SYSTEM NEWQuestion2V_CNV_V2 (* System Configuration *)
  (* Standard: 61499-1 *)
  (* Version 0.4, 2009-03-05, JHC, Holobloc Inc., Deleted Application. *)
  (* Version 0.3, 2003-12-05, JHC, Rockwell Automation, Renamed from NEWSYSTEM. *)
  (* Version 0.2, 2002-11-05, JHC, Rockwell Automation, Fixed missing (empty) FBD in Application. *)
  (* Version 0.1, 2002-01-17, JHC, Rockwell Automation, Minor cleanup *)
  (* Version 0.0, 2000-05-27, JHC, Rockwell Automation *)
  DEVICE HMI : FRAME_DEVICE(GRID := [6,1], BOUNDS := [810,10,300,300])
    RESOURCE reset : PANEL_RESOURCE
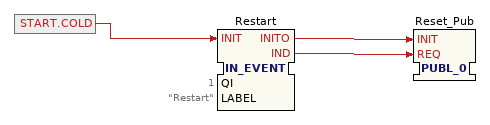
      FBS
        Restart : IN_EVENT(QI := 1, LABEL := "Restart");
        Reset_Pub : PUBL_0;
      END_FBS
      EVENT_CONNECTIONS
        START.COLD TO Restart.INIT;
        Restart.INITO TO Reset_Pub.INIT;
        Restart.IND TO Reset_Pub.REQ;
      END_CONNECTIONS
    END_RESOURCE
    RESOURCE motor_1 : PANEL_RESOURCE
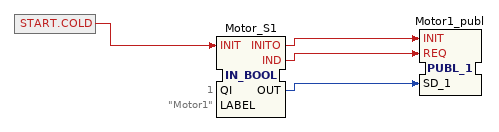
      FBS
        Motor_S1 : IN_BOOL(QI := 1, LABEL := "Motor1");
        Motor1_publ : PUBL_1;
      END_FBS
      EVENT_CONNECTIONS
        START.COLD TO Motor_S1.INIT;
        Motor_S1.INITO TO Motor1_publ.INIT;
        Motor_S1.IND TO Motor1_publ.REQ;
      END_CONNECTIONS
      DATA_CONNECTIONS
        Motor_S1.OUT TO Motor1_publ.SD_1;
      END_CONNECTIONS
    END_RESOURCE
    RESOURCE motor2 : PANEL_RESOURCE
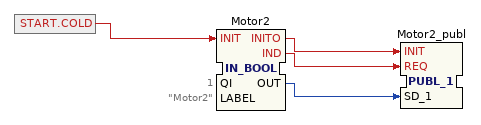
      FBS
        Motor2 : IN_BOOL(QI := 1, LABEL := "Motor2");
        Motor2_publ : PUBL_1;
      END_FBS
      EVENT_CONNECTIONS
        START.COLD TO Motor2.INIT;
        Motor2.INITO TO Motor2_publ.INIT;
        Motor2.IND TO Motor2_publ.REQ;
      END_CONNECTIONS
      DATA_CONNECTIONS
        Motor2.OUT TO Motor2_publ.SD_1;
      END_CONNECTIONS
    END_RESOURCE
    RESOURCE motor3_red : PANEL_RESOURCE
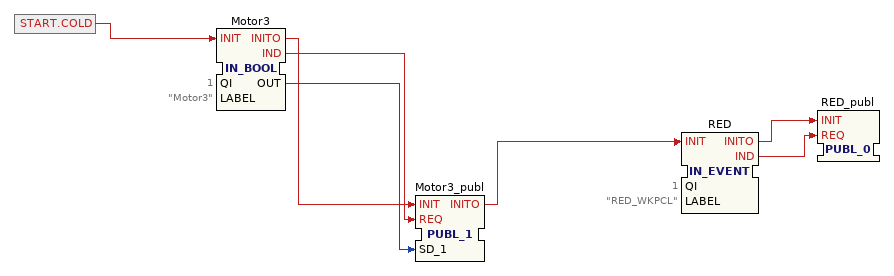
      FBS
        Motor3_publ : PUBL_1;
        Motor3 : IN_BOOL(QI := 1, LABEL := "Motor3");
        RED : IN_EVENT(QI := 1, LABEL := "RED_WKPCL");
        RED_publ : PUBL_0;
      END_FBS
      EVENT_CONNECTIONS
        START.COLD TO Motor3.INIT;
        Motor3.INITO TO Motor3_publ.INIT;
        Motor3.IND TO Motor3_publ.REQ;
        Motor3_publ.INITO TO RED.INIT;
        RED.INITO TO RED_publ.INIT;
        RED.IND TO RED_publ.REQ;
      END_CONNECTIONS
      DATA_CONNECTIONS
        Motor3.OUT TO Motor3_publ.SD_1;
      END_CONNECTIONS
    END_RESOURCE
    RESOURCE motor4_yellow : PANEL_RESOURCE
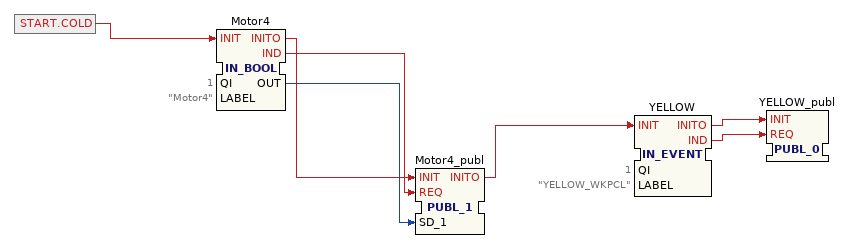
      FBS
        Motor4_publ : PUBL_1;
        Motor4 : IN_BOOL(QI := 1, LABEL := "Motor4");
        YELLOW : IN_EVENT(QI := 1, LABEL := "YELLOW_WKPCL");
        YELLOW_publ : PUBL_0;
      END_FBS
      EVENT_CONNECTIONS
        START.COLD TO Motor4.INIT;
        Motor4.INITO TO Motor4_publ.INIT;
        Motor4.IND TO Motor4_publ.REQ;
        Motor4_publ.INITO TO YELLOW.INIT;
        YELLOW.INITO TO YELLOW_publ.INIT;
        YELLOW.IND TO YELLOW_publ.REQ;
      END_CONNECTIONS
      DATA_CONNECTIONS
        Motor4.OUT TO Motor4_publ.SD_1;
      END_CONNECTIONS
    END_RESOURCE
    RESOURCE motor5_blue : PANEL_RESOURCE
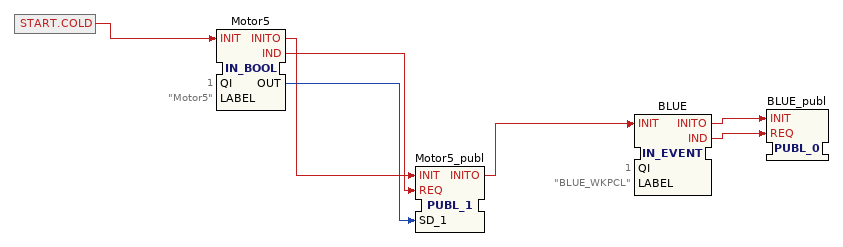
      FBS
        Motor5_publ : PUBL_1;
        Motor5 : IN_BOOL(QI := 1, LABEL := "Motor5");
        BLUE : IN_EVENT(QI := 1, LABEL := "BLUE_WKPCL");
        BLUE_publ : PUBL_0;
      END_FBS
      EVENT_CONNECTIONS
        START.COLD TO Motor5.INIT;
        Motor5.INITO TO Motor5_publ.INIT;
        Motor5.IND TO Motor5_publ.REQ;
        Motor5_publ.INITO TO BLUE.INIT;
        BLUE.INITO TO BLUE_publ.INIT;
        BLUE.IND TO BLUE_publ.REQ;
      END_CONNECTIONS
      DATA_CONNECTIONS
        Motor5.OUT TO Motor5_publ.SD_1;
      END_CONNECTIONS
    END_RESOURCE
  END_DEVICE
  DEVICE VIEW : FRAME_DEVICE(BOUNDS := [10,10,500,700], GRID := [1,1])
    RESOURCE CNV : PANEL_RESOURCE
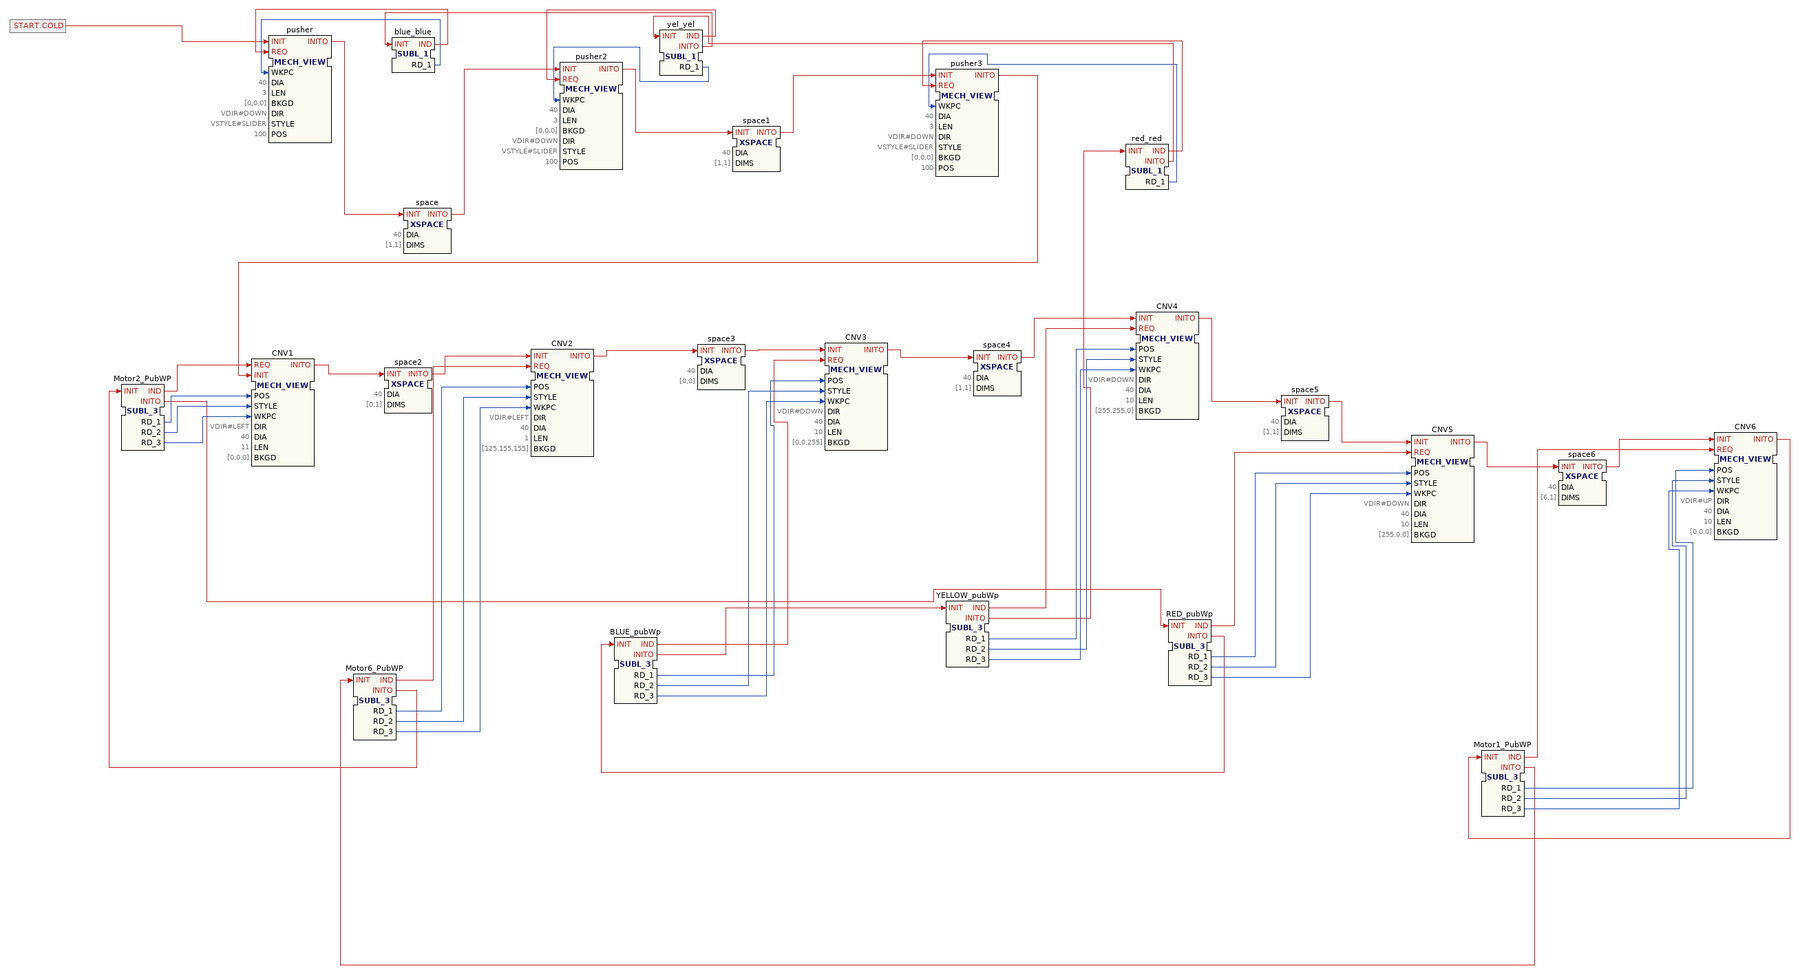
      FBS
        CNV1 : MECH_VIEW(DIR := VDIR#LEFT, DIA := 40, LEN := 11, BKGD := [0,0,0]);
        CNV2 : MECH_VIEW(DIR := VDIR#LEFT, DIA := 40, LEN := 1, BKGD := [125,155,155]);
        CNV3 : MECH_VIEW(DIR := VDIR#DOWN, DIA := 40, LEN := 10, BKGD := [0,0,255]);
        CNV4 : MECH_VIEW(DIR := VDIR#DOWN, DIA := 40, LEN := 10, BKGD := [255,255,0]);
        CNV5 : MECH_VIEW(DIR := VDIR#DOWN, DIA := 40, LEN := 10, BKGD := [255,0,0]);
        CNV6 : MECH_VIEW(DIR := VDIR#UP, DIA := 40, LEN := 10, BKGD := [0,0,0]);
        space2 : XSPACE(DIA := 40, DIMS := [0,1]);
        space3 : XSPACE(DIA := 40, DIMS := [0,0]);
        space4 : XSPACE(DIA := 40, DIMS := [1,1]);
        space5 : XSPACE(DIA := 40, DIMS := [1,1]);
        space6 : XSPACE(DIA := 40, DIMS := [6,1]);
        space : XSPACE(DIA := 40, DIMS := [1,1]);
        space1 : XSPACE(DIA := 40, DIMS := [1,1]);
        Motor1_PubWP : SUBL_3;
        Motor6_PubWP : SUBL_3;
        Motor2_PubWP : SUBL_3;
        BLUE_pubWp : SUBL_3;
        YELLOW_pubWp : SUBL_3;
        RED_pubWp : SUBL_3;
        pusher : MECH_VIEW(DIA := 40, LEN := 3, BKGD := [0,0,0], DIR := VDIR#DOWN, STYLE := VSTYLE#SLIDER, POS := 100);
        pusher2 : MECH_VIEW(DIA := 40, LEN := 3, BKGD := [0,0,0], DIR := VDIR#DOWN, STYLE := VSTYLE#SLIDER, POS := 100);
        pusher3 : MECH_VIEW(DIA := 40, LEN := 3, DIR := VDIR#DOWN, STYLE := VSTYLE#SLIDER, BKGD := [0,0,0], POS := 100);
        red_red : SUBL_1;
        yel_yel : SUBL_1;
        blue_blue : SUBL_1;
      END_FBS
      EVENT_CONNECTIONS
        CNV1.INITO TO space2.INIT;
        space2.INITO TO CNV2.INIT;
        CNV2.INITO TO space3.INIT;
        space3.INITO TO CNV3.INIT;
        CNV3.INITO TO space4.INIT;
        space4.INITO TO CNV4.INIT;
        CNV4.INITO TO space5.INIT;
        space5.INITO TO CNV5.INIT;
        CNV5.INITO TO space6.INIT;
        space6.INITO TO CNV6.INIT;
        CNV6.INITO TO Motor1_PubWP.INIT;
        Motor1_PubWP.IND TO CNV6.REQ;
        Motor1_PubWP.INITO TO Motor6_PubWP.INIT;
        Motor6_PubWP.IND TO CNV2.REQ;
        Motor6_PubWP.INITO TO Motor2_PubWP.INIT;
        Motor2_PubWP.IND TO CNV1.REQ;
        BLUE_pubWp.IND TO CNV3.REQ;
        BLUE_pubWp.INITO TO YELLOW_pubWp.INIT;
        YELLOW_pubWp.IND TO CNV4.REQ;
        RED_pubWp.IND TO CNV5.REQ;
        Motor2_PubWP.INITO TO RED_pubWp.INIT;
        RED_pubWp.INITO TO BLUE_pubWp.INIT;
        START.COLD TO pusher.INIT;
        pusher.INITO TO space.INIT;
        space.INITO TO pusher2.INIT;
        pusher2.INITO TO space1.INIT;
        space1.INITO TO pusher3.INIT;
        pusher3.INITO TO CNV1.INIT;
        red_red.IND TO pusher3.REQ;
        YELLOW_pubWp.INITO TO red_red.INIT;
        red_red.INITO TO yel_yel.INIT;
        yel_yel.IND TO pusher2.REQ;
        yel_yel.INITO TO blue_blue.INIT;
        blue_blue.IND TO pusher.REQ;
      END_CONNECTIONS
      DATA_CONNECTIONS
        Motor1_PubWP.RD_1 TO CNV6.POS;
        Motor1_PubWP.RD_2 TO CNV6.STYLE;
        Motor1_PubWP.RD_3 TO CNV6.WKPC;
        Motor6_PubWP.RD_1 TO CNV2.POS;
        Motor6_PubWP.RD_2 TO CNV2.STYLE;
        Motor6_PubWP.RD_3 TO CNV2.WKPC;
        Motor2_PubWP.RD_1 TO CNV1.POS;
        Motor2_PubWP.RD_2 TO CNV1.STYLE;
        Motor2_PubWP.RD_3 TO CNV1.WKPC;
        BLUE_pubWp.RD_1 TO CNV3.POS;
        BLUE_pubWp.RD_2 TO CNV3.STYLE;
        BLUE_pubWp.RD_3 TO CNV3.WKPC;
        YELLOW_pubWp.RD_1 TO CNV4.POS;
        YELLOW_pubWp.RD_2 TO CNV4.STYLE;
        YELLOW_pubWp.RD_3 TO CNV4.WKPC;
        RED_pubWp.RD_1 TO CNV5.POS;
        RED_pubWp.RD_2 TO CNV5.STYLE;
        RED_pubWp.RD_3 TO CNV5.WKPC;
        red_red.RD_1 TO pusher3.WKPC;
        yel_yel.RD_1 TO pusher2.WKPC;
        blue_blue.RD_1 TO pusher.WKPC;
      END_CONNECTIONS
    END_RESOURCE
  END_DEVICE
  DEVICE MODEL : FRAME_DEVICE(BOUNDS := [0,0,0,0], GRID := [1,1])
    RESOURCE CLK : PANEL_RESOURCE
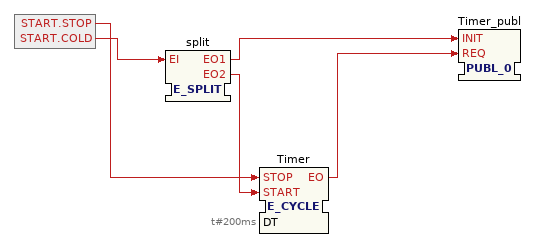
      FBS
        Timer : E_CYCLE(DT := t#200ms);
        Timer_publ : PUBL_0;
        split : E_SPLIT;
      END_FBS
      EVENT_CONNECTIONS
        START.STOP TO Timer.STOP;
        START.COLD TO split.EI;
        split.EO1 TO Timer_publ.INIT;
        split.EO2 TO Timer.START;
        Timer.EO TO Timer_publ.REQ;
      END_CONNECTIONS
    END_RESOURCE
    RESOURCE Motor1 : PANEL_RESOURCE
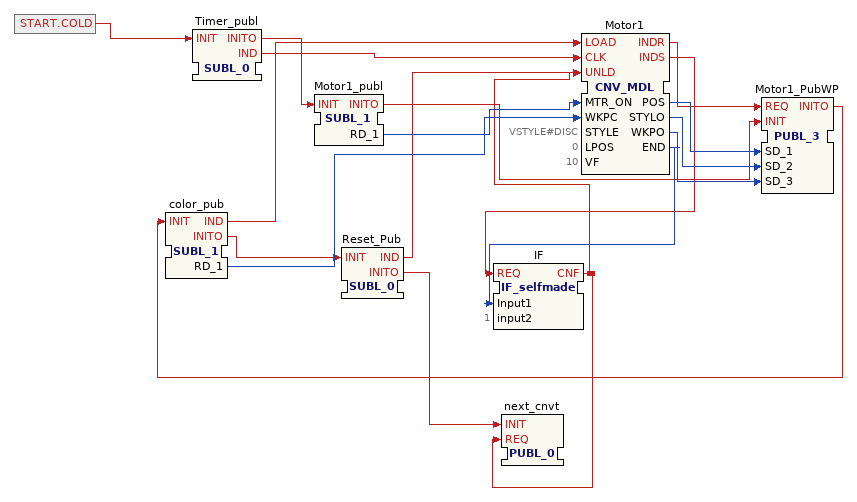
      FBS
        Timer_publ : SUBL_0;
        Motor1_publ : SUBL_1;
        Motor1 : CNV_MDL(STYLE := VSTYLE#DISC, LPOS := 0, VF := 10);
        Motor1_PubWP : PUBL_3;
        color_pub : SUBL_1;
        Reset_Pub : SUBL_0;
        IF : IF_selfmade(input2 := 1);
        next_cnvt : PUBL_0;
      END_FBS
      EVENT_CONNECTIONS
        START.COLD TO Timer_publ.INIT;
        Timer_publ.INITO TO Motor1_publ.INIT;
        Motor1.INDR TO Motor1_PubWP.REQ;
        Motor1_publ.INITO TO Motor1_PubWP.INIT;
        Motor1_PubWP.INITO TO color_pub.INIT;
        color_pub.IND TO Motor1.LOAD;
        Timer_publ.IND TO Motor1.CLK;
        color_pub.INITO TO Reset_Pub.INIT;
        Reset_Pub.IND TO Motor1.UNLD;
        Motor1.INDS TO IF.REQ;
        IF.CNF TO Motor1.UNLD;
        Reset_Pub.INITO TO next_cnvt.INIT;
        IF.CNF TO next_cnvt.REQ;
      END_CONNECTIONS
      DATA_CONNECTIONS
        Motor1_publ.RD_1 TO Motor1.MTR_ON;
        Motor1.POS TO Motor1_PubWP.SD_1;
        Motor1.STYLO TO Motor1_PubWP.SD_2;
        Motor1.WKPO TO Motor1_PubWP.SD_3;
        color_pub.RD_1 TO Motor1.WKPC;
        Motor1.END TO IF.Input1;
      END_CONNECTIONS
    END_RESOURCE
    RESOURCE motor2 : PANEL_RESOURCE
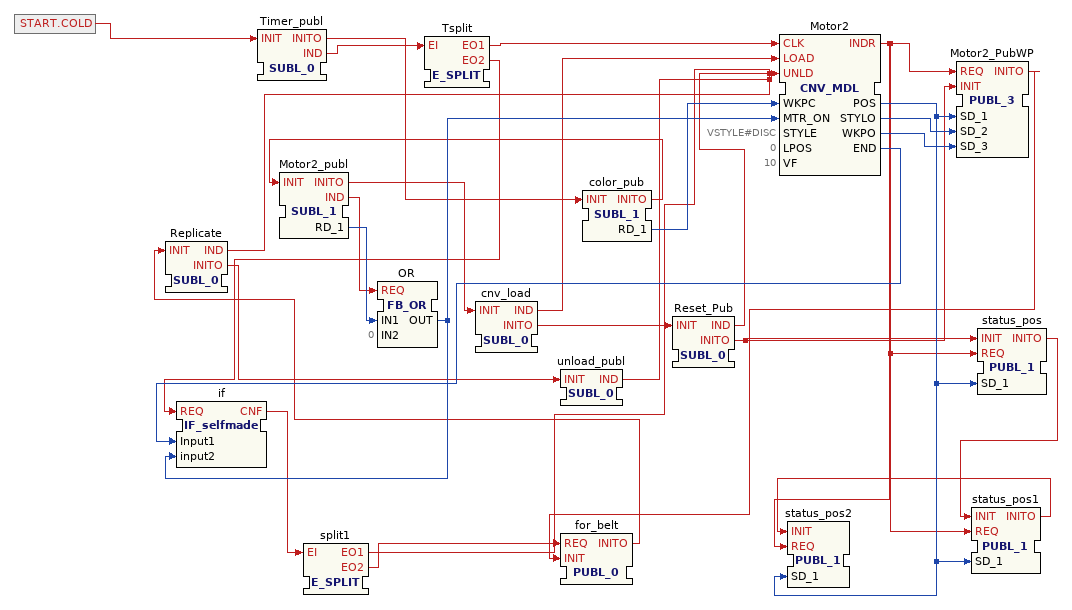
      FBS
        Motor2 : CNV_MDL(STYLE := VSTYLE#DISC, LPOS := 0, VF := 10);
        Timer_publ : SUBL_0;
        Tsplit : E_SPLIT;
        color_pub : SUBL_1;
        Motor2_publ : SUBL_1;
        cnv_load : SUBL_0;
        Motor2_PubWP : PUBL_3;
        Reset_Pub : SUBL_0;
        split1 : E_SPLIT;
        if : IF_selfmade;
        OR : FB_OR(IN2 := 0);
        for_belt : PUBL_0;
        Replicate : SUBL_0;
        unload_publ : SUBL_0;
        status_pos : PUBL_1;
        status_pos1 : PUBL_1;
        status_pos2 : PUBL_1;
      END_FBS
      EVENT_CONNECTIONS
        START.COLD TO Timer_publ.INIT;
        Tsplit.EO1 TO Motor2.CLK;
        color_pub.INITO TO Motor2_publ.INIT;
        Motor2_publ.INITO TO cnv_load.INIT;
        cnv_load.IND TO Motor2.LOAD;
        Timer_publ.INITO TO color_pub.INIT;
        Reset_Pub.IND TO Motor2.UNLD;
        Motor2.INDR TO Motor2_PubWP.REQ;
        Reset_Pub.INITO TO Motor2_PubWP.INIT;
        split1.EO1 TO Motor2.UNLD;
        if.CNF TO split1.EI;
        Motor2_publ.IND TO OR.REQ;
        cnv_load.INITO TO Reset_Pub.INIT;
        Tsplit.EO2 TO if.REQ;
        split1.EO2 TO for_belt.REQ;
        Motor2_PubWP.INITO TO for_belt.INIT;
        Timer_publ.IND TO Tsplit.EI;
        Replicate.IND TO Motor2.UNLD;
        for_belt.INITO TO Replicate.INIT;
        unload_publ.IND TO Motor2.UNLD;
        Replicate.INITO TO unload_publ.INIT;
        Reset_Pub.INITO TO status_pos.INIT;
        Motor2.INDR TO status_pos.REQ;
        status_pos.INITO TO status_pos1.INIT;
        Motor2.INDR TO status_pos1.REQ;
        status_pos1.INITO TO status_pos2.INIT;
        Motor2.INDR TO status_pos2.REQ;
      END_CONNECTIONS
      DATA_CONNECTIONS
        color_pub.RD_1 TO Motor2.WKPC;
        Motor2.POS TO Motor2_PubWP.SD_1;
        Motor2.STYLO TO Motor2_PubWP.SD_2;
        Motor2.WKPO TO Motor2_PubWP.SD_3;
        Motor2_publ.RD_1 TO OR.IN1;
        OR.OUT TO Motor2.MTR_ON;
        OR.OUT TO if.input2;
        Motor2.END TO if.Input1;
        Motor2.POS TO status_pos.SD_1;
        Motor2.POS TO status_pos1.SD_1;
        Motor2.POS TO status_pos2.SD_1;
      END_CONNECTIONS
    END_RESOURCE
    RESOURCE motor3_red : PANEL_RESOURCE
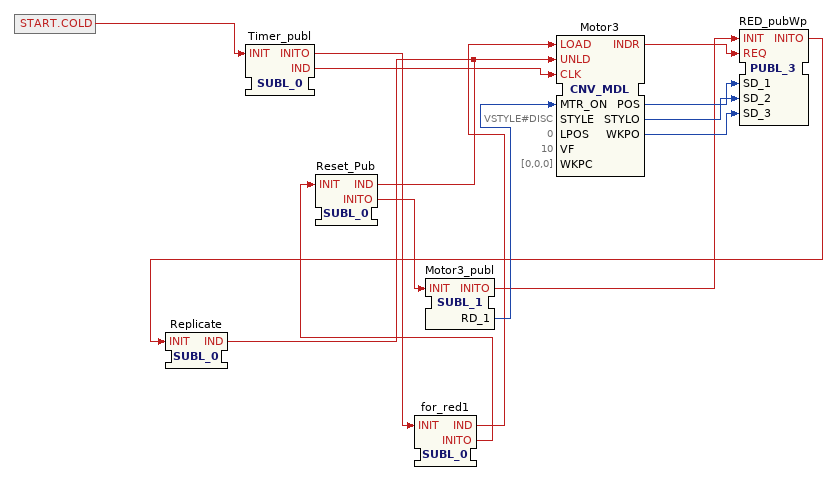
      FBS
        Timer_publ : SUBL_0;
        Motor3 : CNV_MDL(STYLE := VSTYLE#DISC, LPOS := 0, VF := 10, WKPC := [0,0,0]);
        for_red1 : SUBL_0;
        Reset_Pub : SUBL_0;
        Motor3_publ : SUBL_1;
        RED_pubWp : PUBL_3;
        Replicate : SUBL_0;
      END_FBS
      EVENT_CONNECTIONS
        START.COLD TO Timer_publ.INIT;
        Timer_publ.INITO TO for_red1.INIT;
        for_red1.IND TO Motor3.LOAD;
        for_red1.INITO TO Reset_Pub.INIT;
        Reset_Pub.IND TO Motor3.UNLD;
        Reset_Pub.INITO TO Motor3_publ.INIT;
        Motor3_publ.INITO TO RED_pubWp.INIT;
        Motor3.INDR TO RED_pubWp.REQ;
        Timer_publ.IND TO Motor3.CLK;
        RED_pubWp.INITO TO Replicate.INIT;
        Replicate.IND TO Motor3.UNLD;
      END_CONNECTIONS
      DATA_CONNECTIONS
        Motor3_publ.RD_1 TO Motor3.MTR_ON;
        Motor3.POS TO RED_pubWp.SD_1;
        Motor3.STYLO TO RED_pubWp.SD_2;
        Motor3.WKPO TO RED_pubWp.SD_3;
      END_CONNECTIONS
    END_RESOURCE
    RESOURCE motor4_yellow : PANEL_RESOURCE
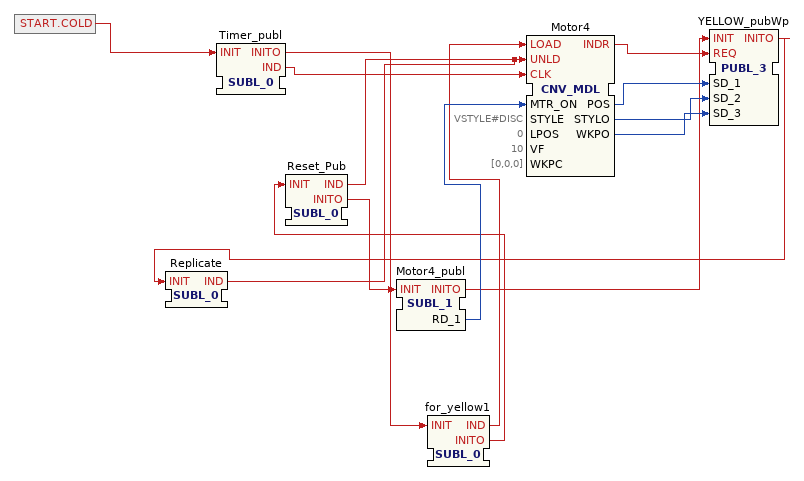
      FBS
        Timer_publ : SUBL_0;
        Motor4 : CNV_MDL(STYLE := VSTYLE#DISC, LPOS := 0, VF := 10, WKPC := [0,0,0]);
        for_yellow1 : SUBL_0;
        Reset_Pub : SUBL_0;
        Motor4_publ : SUBL_1;
        YELLOW_pubWp : PUBL_3;
        Replicate : SUBL_0;
      END_FBS
      EVENT_CONNECTIONS
        START.COLD TO Timer_publ.INIT;
        Timer_publ.INITO TO for_yellow1.INIT;
        for_yellow1.IND TO Motor4.LOAD;
        for_yellow1.INITO TO Reset_Pub.INIT;
        Reset_Pub.IND TO Motor4.UNLD;
        Reset_Pub.INITO TO Motor4_publ.INIT;
        Motor4_publ.INITO TO YELLOW_pubWp.INIT;
        Motor4.INDR TO YELLOW_pubWp.REQ;
        Timer_publ.IND TO Motor4.CLK;
        YELLOW_pubWp.INITO TO Replicate.INIT;
        Replicate.IND TO Motor4.UNLD;
      END_CONNECTIONS
      DATA_CONNECTIONS
        Motor4_publ.RD_1 TO Motor4.MTR_ON;
        Motor4.POS TO YELLOW_pubWp.SD_1;
        Motor4.STYLO TO YELLOW_pubWp.SD_2;
        Motor4.WKPO TO YELLOW_pubWp.SD_3;
      END_CONNECTIONS
    END_RESOURCE
    RESOURCE motor5_blue : PANEL_RESOURCE
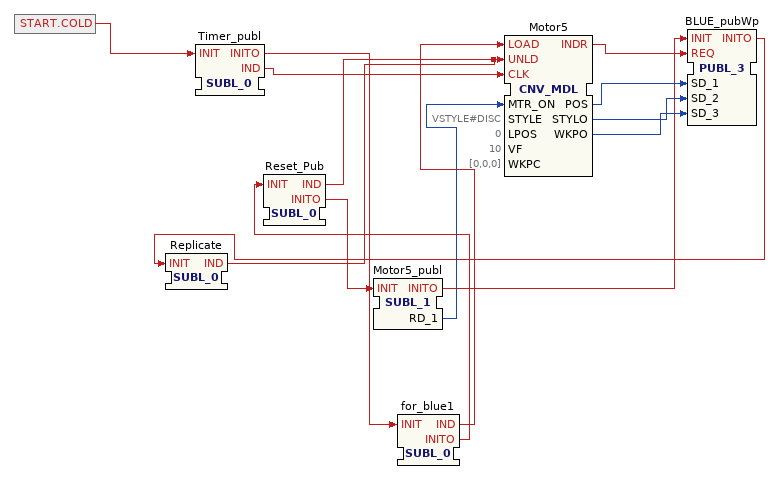
      FBS
        Timer_publ : SUBL_0;
        Motor5 : CNV_MDL(STYLE := VSTYLE#DISC, LPOS := 0, VF := 10, WKPC := [0,0,0]);
        for_blue1 : SUBL_0;
        Reset_Pub : SUBL_0;
        Motor5_publ : SUBL_1;
        BLUE_pubWp : PUBL_3;
        Replicate : SUBL_0;
      END_FBS
      EVENT_CONNECTIONS
        START.COLD TO Timer_publ.INIT;
        Timer_publ.INITO TO for_blue1.INIT;
        for_blue1.IND TO Motor5.LOAD;
        for_blue1.INITO TO Reset_Pub.INIT;
        Reset_Pub.IND TO Motor5.UNLD;
        Reset_Pub.INITO TO Motor5_publ.INIT;
        Motor5_publ.INITO TO BLUE_pubWp.INIT;
        Motor5.INDR TO BLUE_pubWp.REQ;
        Timer_publ.IND TO Motor5.CLK;
        BLUE_pubWp.INITO TO Replicate.INIT;
        Replicate.IND TO Motor5.UNLD;
      END_CONNECTIONS
      DATA_CONNECTIONS
        Motor5_publ.RD_1 TO Motor5.MTR_ON;
        Motor5.POS TO BLUE_pubWp.SD_1;
        Motor5.STYLO TO BLUE_pubWp.SD_2;
        Motor5.WKPO TO BLUE_pubWp.SD_3;
      END_CONNECTIONS
    END_RESOURCE
    RESOURCE motor6_turntable : PANEL_RESOURCE
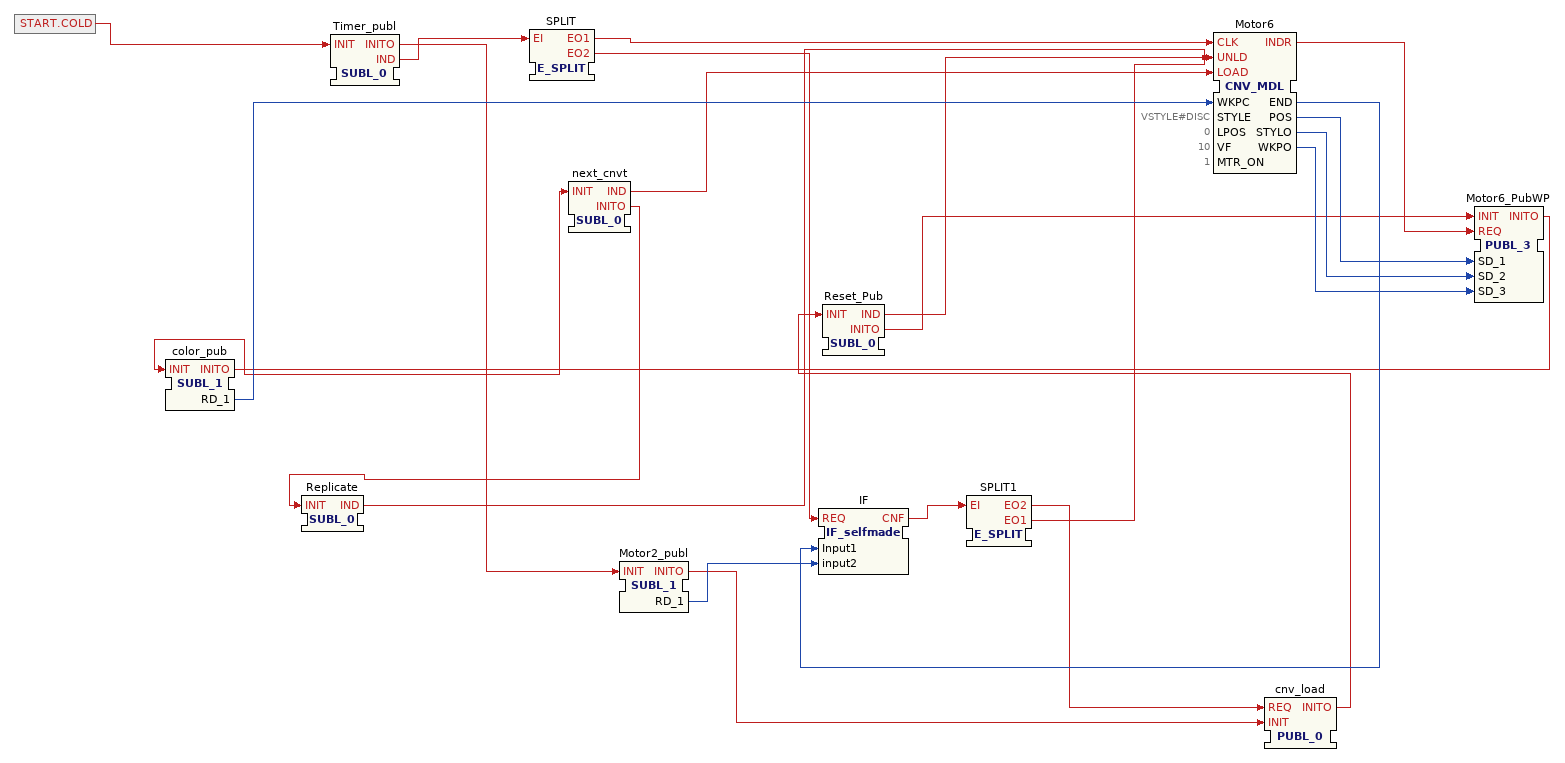
      FBS
        Motor6 : CNV_MDL(STYLE := VSTYLE#DISC, LPOS := 0, VF := 10, MTR_ON := 1);
        Timer_publ : SUBL_0;
        SPLIT : E_SPLIT;
        Motor2_publ : SUBL_1;
        IF : IF_selfmade;
        SPLIT1 : E_SPLIT;
        cnv_load : PUBL_0;
        Reset_Pub : SUBL_0;
        Motor6_PubWP : PUBL_3;
        color_pub : SUBL_1;
        next_cnvt : SUBL_0;
        Replicate : SUBL_0;
      END_FBS
      EVENT_CONNECTIONS
        START.COLD TO Timer_publ.INIT;
        SPLIT.EO1 TO Motor6.CLK;
        Timer_publ.INITO TO Motor2_publ.INIT;
        SPLIT.EO2 TO IF.REQ;
        IF.CNF TO SPLIT1.EI;
        SPLIT1.EO2 TO cnv_load.REQ;
        Motor2_publ.INITO TO cnv_load.INIT;
        cnv_load.INITO TO Reset_Pub.INIT;
        Reset_Pub.IND TO Motor6.UNLD;
        Reset_Pub.INITO TO Motor6_PubWP.INIT;
        Motor6.INDR TO Motor6_PubWP.REQ;
        Motor6_PubWP.INITO TO color_pub.INIT;
        color_pub.INITO TO next_cnvt.INIT;
        next_cnvt.IND TO Motor6.LOAD;
        Timer_publ.IND TO SPLIT.EI;
        SPLIT1.EO1 TO Motor6.UNLD;
        next_cnvt.INITO TO Replicate.INIT;
        Replicate.IND TO Motor6.UNLD;
      END_CONNECTIONS
      DATA_CONNECTIONS
        Motor6.END TO IF.Input1;
        Motor2_publ.RD_1 TO IF.input2;
        Motor6.POS TO Motor6_PubWP.SD_1;
        Motor6.STYLO TO Motor6_PubWP.SD_2;
        Motor6.WKPO TO Motor6_PubWP.SD_3;
        color_pub.RD_1 TO Motor6.WKPC;
      END_CONNECTIONS
    END_RESOURCE
  END_DEVICE
  DEVICE CONTROL : FRAME_DEVICE(BOUNDS := [0,0,0,0], GRID := [1,1])
    RESOURCE Color_control : PANEL_RESOURCE
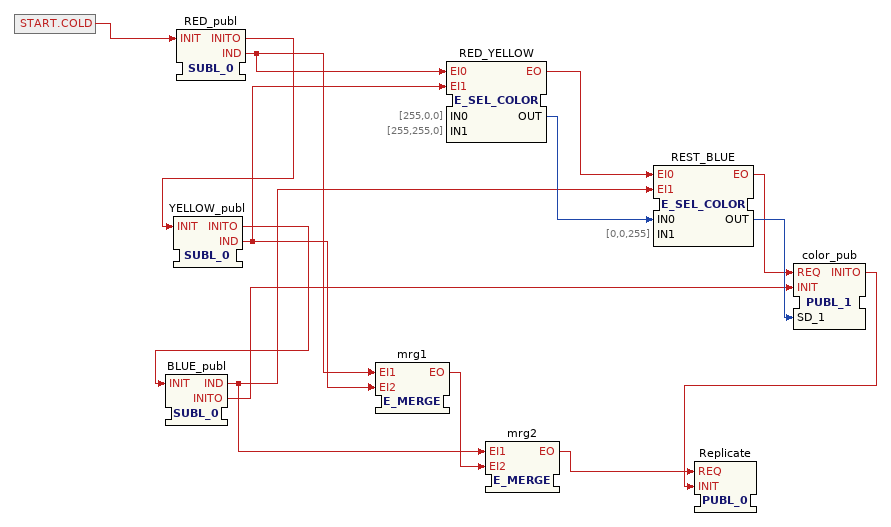
      FBS
        RED_publ : SUBL_0;
        YELLOW_publ : SUBL_0;
        BLUE_publ : SUBL_0;
        RED_YELLOW : E_SEL_COLOR(IN0 := [255,0,0], IN1 := [255,255,0]);
        REST_BLUE : E_SEL_COLOR(IN1 := [0,0,255]);
        color_pub : PUBL_1;
        mrg1 : E_MERGE;
        mrg2 : E_MERGE;
        Replicate : PUBL_0;
      END_FBS
      EVENT_CONNECTIONS
        START.COLD TO RED_publ.INIT;
        RED_publ.INITO TO YELLOW_publ.INIT;
        YELLOW_publ.INITO TO BLUE_publ.INIT;
        RED_publ.IND TO RED_YELLOW.EI0;
        YELLOW_publ.IND TO RED_YELLOW.EI1;
        RED_YELLOW.EO TO REST_BLUE.EI0;
        BLUE_publ.IND TO REST_BLUE.EI1;
        REST_BLUE.EO TO color_pub.REQ;
        BLUE_publ.INITO TO color_pub.INIT;
        RED_publ.IND TO mrg1.EI1;
        YELLOW_publ.IND TO mrg1.EI2;
        BLUE_publ.IND TO mrg2.EI1;
        mrg1.EO TO mrg2.EI2;
        mrg2.EO TO Replicate.REQ;
        color_pub.INITO TO Replicate.INIT;
      END_CONNECTIONS
      DATA_CONNECTIONS
        RED_YELLOW.OUT TO REST_BLUE.IN0;
        REST_BLUE.OUT TO color_pub.SD_1;
      END_CONNECTIONS
    END_RESOURCE
    RESOURCE PUSHER : PANEL_RESOURCE
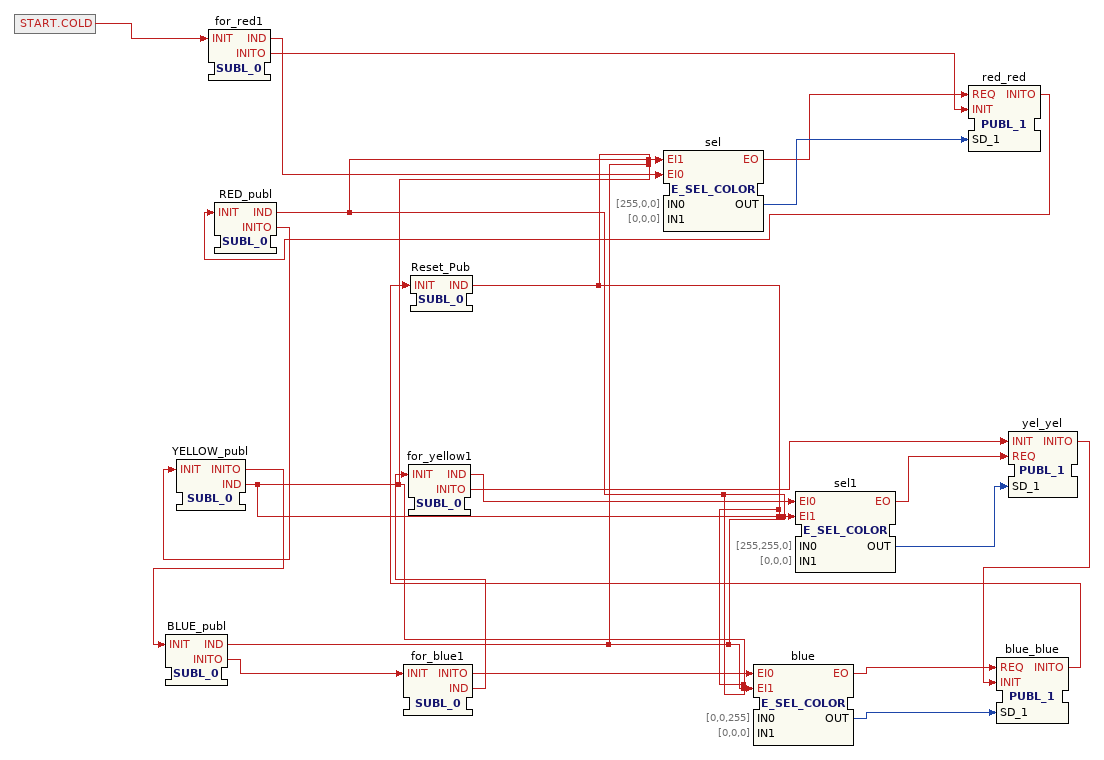
      FBS
        sel : E_SEL_COLOR(IN0 := [255,0,0], IN1 := [0,0,0]);
        red_red : PUBL_1;
        RED_publ : SUBL_0;
        for_red1 : SUBL_0;
        YELLOW_publ : SUBL_0;
        BLUE_publ : SUBL_0;
        for_yellow1 : SUBL_0;
        for_blue1 : SUBL_0;
        sel1 : E_SEL_COLOR(IN0 := [255,255,0], IN1 := [0,0,0]);
        blue : E_SEL_COLOR(IN0 := [0,0,255], IN1 := [0,0,0]);
        yel_yel : PUBL_1;
        blue_blue : PUBL_1;
        Reset_Pub : SUBL_0;
      END_FBS
      EVENT_CONNECTIONS
        sel.EO TO red_red.REQ;
        red_red.INITO TO RED_publ.INIT;
        RED_publ.IND TO sel.EI1;
        START.COLD TO for_red1.INIT;
        for_red1.IND TO sel.EI0;
        for_red1.INITO TO red_red.INIT;
        RED_publ.INITO TO YELLOW_publ.INIT;
        YELLOW_publ.INITO TO BLUE_publ.INIT;
        YELLOW_publ.IND TO sel.EI1;
        BLUE_publ.IND TO sel.EI1;
        BLUE_publ.INITO TO for_blue1.INIT;
        for_blue1.INITO TO for_yellow1.INIT;
        for_yellow1.IND TO sel1.EI0;
        YELLOW_publ.IND TO sel1.EI1;
        BLUE_publ.IND TO sel1.EI1;
        RED_publ.IND TO sel1.EI1;
        for_blue1.IND TO blue.EI0;
        YELLOW_publ.IND TO blue.EI1;
        BLUE_publ.IND TO blue.EI1;
        RED_publ.IND TO blue.EI1;
        for_yellow1.INITO TO yel_yel.INIT;
        sel1.EO TO yel_yel.REQ;
        blue.EO TO blue_blue.REQ;
        yel_yel.INITO TO blue_blue.INIT;
        blue_blue.INITO TO Reset_Pub.INIT;
        Reset_Pub.IND TO sel.EI1;
        Reset_Pub.IND TO sel1.EI1;
        Reset_Pub.IND TO blue.EI1;
      END_CONNECTIONS
      DATA_CONNECTIONS
        sel.OUT TO red_red.SD_1;
        sel1.OUT TO yel_yel.SD_1;
        blue.OUT TO blue_blue.SD_1;
      END_CONNECTIONS
    END_RESOURCE
    RESOURCE unload : PANEL_RESOURCE
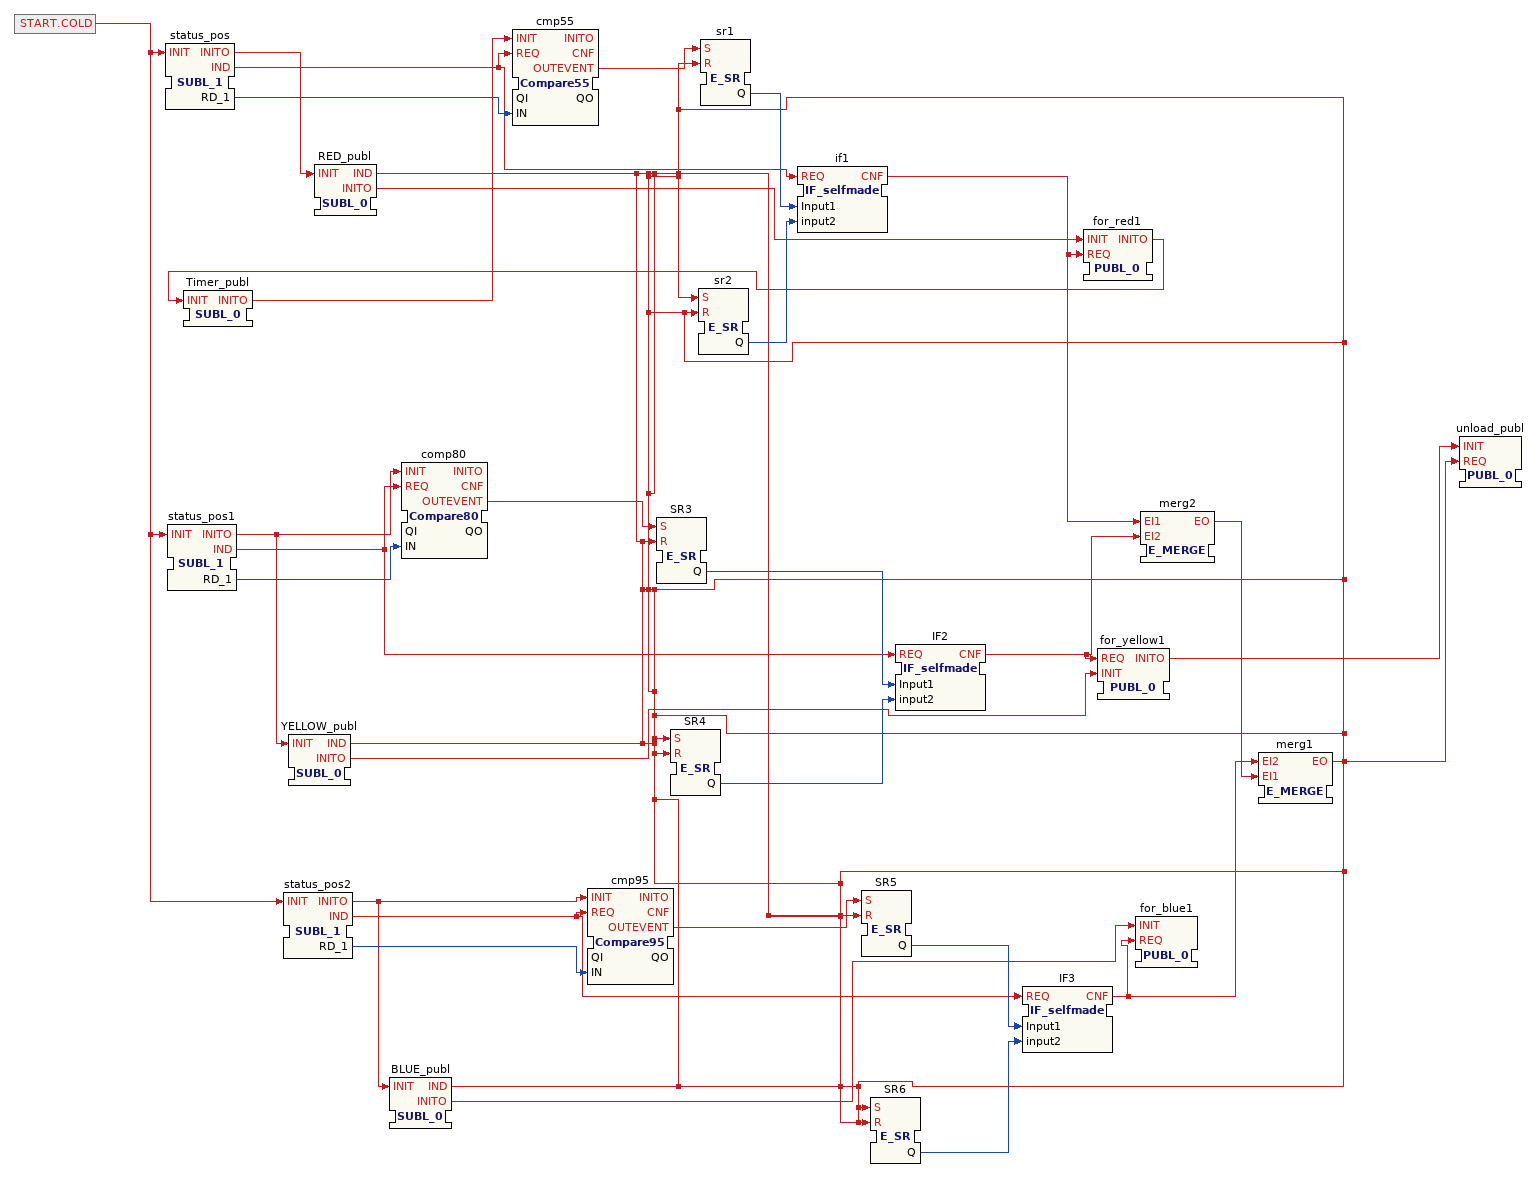
      FBS
        RED_publ : SUBL_0;
        sr1 : E_SR;
        sr2 : E_SR;
        if1 : IF_selfmade;
        Timer_publ : SUBL_0;
        status_pos : SUBL_1;
        cmp55 : Compare55;
        for_red1 : PUBL_0;
        YELLOW_publ : SUBL_0;
        comp80 : Compare80;
        status_pos1 : SUBL_1;
        SR3 : E_SR;
        SR4 : E_SR;
        IF2 : IF_selfmade;
        for_yellow1 : PUBL_0;
        status_pos2 : SUBL_1;
        BLUE_publ : SUBL_0;
        cmp95 : Compare95;
        SR5 : E_SR;
        SR6 : E_SR;
        IF3 : IF_selfmade;
        for_blue1 : PUBL_0;
        merg1 : E_MERGE;
        merg2 : E_MERGE;
        unload_publ : PUBL_0;
      END_FBS
      EVENT_CONNECTIONS
        RED_publ.IND TO sr2.S;
        START.COLD TO status_pos.INIT;
        status_pos.INITO TO RED_publ.INIT;
        Timer_publ.INITO TO cmp55.INIT;
        status_pos.IND TO cmp55.REQ;
        cmp55.OUTEVENT TO sr1.S;
        RED_publ.INITO TO for_red1.INIT;
        if1.CNF TO for_red1.REQ;
        for_red1.INITO TO Timer_publ.INIT;
        status_pos.IND TO if1.REQ;
        START.COLD TO status_pos1.INIT;
        status_pos1.INITO TO YELLOW_publ.INIT;
        status_pos1.INITO TO comp80.INIT;
        status_pos1.IND TO comp80.REQ;
        comp80.OUTEVENT TO SR3.S;
        YELLOW_publ.IND TO SR4.S;
        status_pos1.IND TO IF2.REQ;
        IF2.CNF TO for_yellow1.REQ;
        YELLOW_publ.INITO TO for_yellow1.INIT;
        START.COLD TO status_pos2.INIT;
        status_pos2.INITO TO BLUE_publ.INIT;
        status_pos2.INITO TO cmp95.INIT;
        status_pos2.IND TO cmp95.REQ;
        cmp95.OUTEVENT TO SR5.S;
        BLUE_publ.IND TO SR6.S;
        status_pos2.IND TO IF3.REQ;
        BLUE_publ.INITO TO for_blue1.INIT;
        IF3.CNF TO for_blue1.REQ;
        if1.CNF TO merg2.EI1;
        IF2.CNF TO merg2.EI2;
        IF3.CNF TO merg1.EI2;
        merg2.EO TO merg1.EI1;
        merg1.EO TO sr1.R;
        merg1.EO TO sr2.R;
        merg1.EO TO SR3.R;
        merg1.EO TO SR4.R;
        merg1.EO TO SR5.R;
        merg1.EO TO SR6.R;
        for_yellow1.INITO TO unload_publ.INIT;
        merg1.EO TO unload_publ.REQ;
        YELLOW_publ.IND TO sr1.R;
        YELLOW_publ.IND TO sr2.R;
        YELLOW_publ.IND TO SR5.R;
        YELLOW_publ.IND TO SR6.R;
        BLUE_publ.IND TO SR4.R;
        BLUE_publ.IND TO SR3.R;
        BLUE_publ.IND TO sr2.R;
        BLUE_publ.IND TO sr1.R;
        RED_publ.IND TO SR3.R;
        RED_publ.IND TO SR4.R;
        RED_publ.IND TO SR5.R;
        RED_publ.IND TO SR6.R;
        RED_publ.IND TO sr1.R;
        YELLOW_publ.IND TO SR3.R;
        BLUE_publ.IND TO SR5.R;
      END_CONNECTIONS
      DATA_CONNECTIONS
        sr1.Q TO if1.Input1;
        sr2.Q TO if1.input2;
        status_pos.RD_1 TO cmp55.IN;
        status_pos1.RD_1 TO comp80.IN;
        SR3.Q TO IF2.Input1;
        SR4.Q TO IF2.input2;
        status_pos2.RD_1 TO cmp95.IN;
        SR5.Q TO IF3.Input1;
        SR6.Q TO IF3.input2;
      END_CONNECTIONS
    END_RESOURCE
  END_DEVICE
END_SYSTEM
